// TwinCAT 3 PLC project OpenWeatherMap
// Title: OpenWeatherMap
// Company: Stefan Besler
// Author: Stefan Besler and contributors
// ProjectVersion: 1.0.0
// ProgramVersion: 3.1.4023.0
// libraries:
//   Tc2_Standard, * (Beckhoff Automation GmbH)
//   Tc2_System, * (Beckhoff Automation GmbH)
//   Testbench, * (Zeugwerk GmbH)
// project tree:
//   / OpenWeatherMapClient.TcPOU
//   _DataTypes/ OpenWeatherMapRequest.TcDUT, OpenWeatherMapResponse.TcDUT
//   _Tests/ OpenWeatherMapClientTest.TcPOU (not stored)

// ---- _DataTypes/OpenWeatherMapRequest.TcDUT
{attribute 'pack_mode' := '1'}
TYPE INTERNAL OpenWeatherMapRequest :
STRUCT
  TokenLength : INT;
  Token : STRING(80);
  ZipCodeLength : INT;
  ZipCode : STRING(9);
  CountryCodeLength : INT;
  CountryCode : STRING(4);  
END_STRUCT
END_TYPE

// ---- _DataTypes/OpenWeatherMapResponse.TcDUT
{attribute 'pack_mode' := '1'}
TYPE INTERNAL OpenWeatherMapResponse :
STRUCT
   {attribute 'hide'}
   Status : INT;
   
   {attribute 'hide'}
   Exception : STRING(255);   
  
   CityName : STRING(255);
   Condition : STRING(255);
   TemperatureInCelsius : LREAL;
   FeelsLikeInCelsius : LREAL;
   PressureInBar : LREAL;
   RelativeHumidityInPercent : LREAL;
   MinimumTemperatureInCelsius : LREAL;
   MaximumTemperatureInCelsius : LREAL;
   SeaLevelPressureInBar : LREAL;
   GroundLevelPressureInBar : LREAL;
   WindSpeedInMeterPerSecond : LREAL;
   WindDirectionInDegree : LREAL;
   WindGustInMeterPerSecond : LREAL;
   CloudinessInPercent : LREAL;
   RainfallLastHourInMillimeter : LREAL;
   RainfallLastThreeHoursInMillimeter : LREAL;
   SnowfallLastHourInMillimeter : LREAL;
   SnowfallLastThreeHoursInMillimeter : LREAL;
   SunriseUtc : LWORD;
   SunsetUtc : LWORD;
   UtcOffsetInMillisecond : LWORD;
   FetchedAtUtc : LWORD;
   MeasuredAtUtc : LWORD;
   CityId : DINT;   
   

END_STRUCT
END_TYPE

// ---- OpenWeatherMapClient.TcPOU
/// This the main class of the library. It represents a OpenWeatherMap app and
/// is tied to a unique API token. When constructing the object it is mandatory to pass
/// an `app-token``.
///
/// Here's a simple example, which requests the current data for 'Innsbruck, AT'.
/// The actual action of sending the notification is triggered by [RequestWeatherByZipCodeAsync](xref:OpenWeatherMap.OpenWeatherMapClient#RequestWeatherByZipCodeAsync).
/// The ´Async´ Suffix in this method indicates that this action has to be waited for by checking for ´NOT _openWeatherMapClient.Busy´ before
/// sending another request.
///
/// ```sti
/// PROGRAM MAIN
/// VAR
///   _send : BOOL; // boolean, which can be triggered to send a message
///   _openWeatherMapClient : OpenWeatherMap.OpenWeatherMapClient('<your_openweathermap_apptoken>'); 
/// END_VAR
/// ```
/// ```std
/// IF _send
/// THEN
///   _send := FALSE;
///   _openWeatherMapClient.RequestWeatherByZipCodeAsync('6020', 'AT');
/// END_IF
///
/// _openWeatherMapClient.Cyclic();
/// ```
{attribute 'conditionalshow_all_locals'}
{attribute 'no_explicit_call' := 'This FB is a CLASS and must be accessed using methods and/or properties'}
{attribute 'hide_all_locals'}
FUNCTION_BLOCK OpenWeatherMapClient
VAR
  _busy : BOOL;
  _error : BOOL;
  _errorMessage : STRING(255);
  
  _request : OpenWeatherMapRequest;
  _response : OpenWeatherMapResponse;
  
  _server : Tc2_System.ADSRDWRTEX;
END_VAR
VAR CONSTANT
  _defaultHost : STRING := '127.0.0.1.1.1';
  _defaultPort : UINT := 25734;
END_VAR

/// This property can be used to check if the client is ready for sending request. If the client is not 
/// ready or an error occurs during sending (e.g. not internet connection, OpenWeatherMap Twincat Service is not running, ...)
/// the property [Error](xref:OpenWeatherMap.OpenWeatherMapClient#Error) returns `true`.
{attribute 'monitoring' := 'call'}
PROPERTY Busy : BOOL
GET
Busy := _busy;
END_GET
SET // PROTECTED
_busy := Busy;

IF _busy
THEN
  _error := FALSE;
END_IF
END_SET
END_PROPERTY

/// This method has to be called cyclically and takes care of the communication with the `OpenWeatherMap Twincat Service`, which is reached 
/// via [Host](xref:OpenWeatherMap.OpenWeatherMapClient#Host) and [Port](xref:OpenWeatherMap.OpenWeatherMapClient#Port).
/// You can use the properties [Busy](xref:OpenWeatherMap.OpenWeatherMapClient#Busy) and [Error](xref:OpenWeatherMap.OpenWeatherMapClient#Error) to check weather an
/// operation was successful (`NOT Busy AND NOT Error`) or failed (`Error`), respectively.
METHOD Cyclic
VAR_INST
  errorTrig : Tc2_Standard.R_TRIG;
END_VAR
IF NOT Busy
THEN
  RETURN;
END_IF

_server(IDXOFFS:=0, 
        WRITELEN:=SIZEOF(_request),
        SRCADDR:=ADR(_request),
        WRTRD:=TRUE, 
        TMOUT:=T#5S,
        ERR=>,
        BUSY=>,
        ERRID=>);
  
IF _server.ERR // fallback to proxy
THEN
  Error := TRUE;
  ErrorMessage := Tc2_Standard.CONCAT('Error Code: ', UDINT_TO_STRING(_server.ERRID));
ELSIF NOT _server.BUSY 
THEN
  Busy := FALSE;

  IF _response.Status = 0
  THEN
    Error := TRUE;
    ErrorMessage := 'No data received';  
  ELSIF _response.Status > 0
  THEN
    Error := TRUE;
    ErrorMessage := _response.Exception;
	END_IF

END_IF
END_METHOD

/// Returns `true` if any error occured when calling an `XXX_Async` method of this object. The details of the error
/// are available by checking the proeprty
{attribute 'monitoring' := 'call'}
PROPERTY Error : BOOL
GET
Error := _error;
END_GET
SET // PROTECTED
_error := Error;

IF _error
THEN
  _busy := FALSE;
END_IF
END_SET
END_PROPERTY

/// Only valid if `Error=TRUE`, returns the explanation why the call of an `XXX_Async` method failed.
{attribute 'monitoring' := 'call'}
PROPERTY ErrorMessage : STRING(255)
GET
IF _error
THEN
  ErrorMessage := _errorMessage;
END_IF
END_GET
SET // PROTECTED
_errorMessage := ErrorMessage;
END_SET
END_PROPERTY

METHOD FB_init : BOOL
VAR_INPUT
	bInitRetains : BOOL; // if TRUE, the retain variables are initialized (warm start / cold start)
	bInCopyCode : BOOL;  // if TRUE, the instance afterwards gets moved into the copy code (online change)
  
  /// The OpenWeatherMap API token
  token : STRING;
END_VAR
THIS^.Token := token;
THIS^.Host := _defaultHost;
THIS^.Port := _defaultPort;

Reset();
END_METHOD

/// Returns the AMS Net Id of the `OpenWeatherMap Twincat Service`. Defaults to localhost
PROPERTY Host : STRING
GET
Host := _server.NETID;
END_GET
SET
_server(WRTRD := FALSE,
       NETID := Host,
       BUSY=>,
       ERR=>,
       ERRID=>);
END_SET
END_PROPERTY

PROPERTY Port : UINT
GET
Port := _server.PORT;
END_GET
SET
_server(WRTRD := FALSE,
       PORT := Port,
       BUSY=>,
       ERR=>,
       ERRID=>);
END_SET
END_PROPERTY

METHOD RequestWeatherByZipCodeAsync
VAR_IN_OUT CONSTANT
  zipCode : STRING(9);
  countryCode : STRING(4);
END_VAR
IF NOT Busy
THEN
  _request.ZipCodeLength := Tc2_Standard.LEN(zipCode);
  _request.ZipCode := zipCode;
  _request.CountryCodeLength := Tc2_Standard.LEN(countryCode);
  _request.CountryCode := countryCode;
  
  _response.Status := 0;
  
  _server(WRTRD := FALSE,
         IDXGRP:=0,
         DESTADDR:=ADR(_response),
         READLEN:=SIZEOF(_response),
         TMOUT:=TIME#10S,
         BUSY=>,
         ERR=>,
         ERRID=>);    
  Busy := TRUE;
ELSE
  Error := TRUE;
  _errorMessage := 'Client can not executed parallel requests!';
END_IF
END_METHOD

/// Resets client to default values
METHOD Reset
VAR
  token : STRING;
  host : STRING;
  port : UINT;  
END_VAR
token := THIS^.Token;
host := THIS^.Host;
port := THIS^.Port;

Tc2_System.MEMSET(ADR(_request), 0, SIZEOF(_request));

THIS^.Token := token;
THIS^.Host := _defaultHost;
THIS^.Port := _defaultPort;
END_METHOD

PROPERTY Token : STRING
GET
Token := _request.Token;
END_GET
SET
_request.Token := Token;
_request.TokenLength := Tc2_Standard.LEN(_request.Token);
END_SET
END_PROPERTY

{attribute 'monitoring' := 'call'}
PROPERTY Weather : REFERENCE TO OpenWeatherMapResponse
GET
IF _busy OR_ELSE _response.Status = 0
THEN
  Weather REF= 0;
  RETURN;
END_IF

Weather REF= _response;
END_GET
END_PROPERTY

END_FUNCTION_BLOCK
